// Mitsubishi GX Works2 project: z03   PLC: Q02/Q02H

PROGRAM MAIN
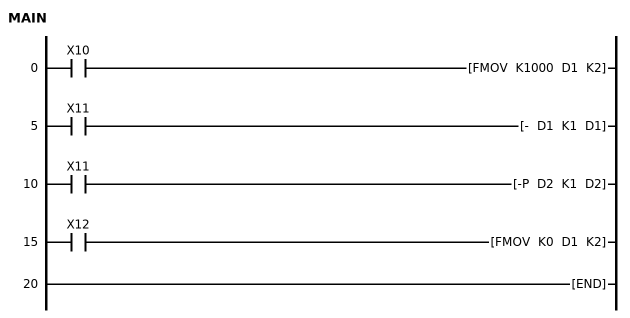
0     LD      X10
      FMOV    K1000 D1 K2
5     LD      X11
      -       D1 K1 D1
10    LD      X11
      -P      D2 K1 D2
15    LD      X12
      FMOV    K0 D1 K2
20    END
END_PROGRAM
